METHOD INTERNAL CreateCommandPayloadLog
VAR_IN_OUT
  /// Robot assignment of function
  AxesGroup : AxesGroup; 
END_VAR
VAR 
  /// internal index for loops
 _idx : DINT;
END_VAR
// Create log entry for Parameter start
CreateLogMessage      ( Timestamp   := AxesGroup.InternalData.SystemTime,
                        MessageType := MessageType.CMD,
                        Severity    := Severity.DEBUG,
                        MessageCode := 0,
                        MessageText := 'Create command payload with the following parameter(s) :');

// Create log entry for Mode
CreateLogMessagePara1 ( Timestamp   := AxesGroup.InternalData.SystemTime,
                        MessageType := MessageType.CMD,
                        Severity    := Severity.DEBUG,
                        MessageCode := 0,
                        MessageText := 'Command.Mode = {1}',
                        Para1       :=  SPLINE_MODE_TO_STRING(_command.Mode));

// Create log entry for SplineID
CreateLogMessagePara1 ( Timestamp   := AxesGroup.InternalData.SystemTime,
                        MessageType := MessageType.CMD,
                        Severity    := Severity.DEBUG,
                        MessageCode := 0,
                        MessageText := 'Command.SplineID = {1}',
                        Para1       :=  SINT_TO_STRING(_command.SplineID));

// Create log entry for SplineData[x]
FOR _idx := 1 TO RobotLibraryParameter.SPLINE_DATA_MAX
DO
  // Create log entry for VelocityRate
  CreateLogMessagePara2 ( Timestamp   := AxesGroup.InternalData.SystemTime,
                          MessageType := MessageType.CMD,
                          Severity    := Severity.DEBUG,
                          MessageCode := 0,
                          MessageText := 'Command.SplineData[{2}].VelocityRate = {1}',
                          Para1       :=  UINT_TO_STRING(_command.SplineData[_idx].VelocityRate),
                          Para2       :=  DINT_TO_STRING(_idx));

  // Create log entry for AccelerationRate
  CreateLogMessagePara2 ( Timestamp   := AxesGroup.InternalData.SystemTime,
                          MessageType := MessageType.CMD,
                          Severity    := Severity.DEBUG,
                          MessageCode := 0,
                          MessageText := 'Command.SplineData[{2}].AccelerationRate = {1}',
                          Para1       :=  UINT_TO_STRING(_command.SplineData[_idx].AccelerationRate),
                          Para2       :=  DINT_TO_STRING(_idx));

  // Create log entry for DecelerationRate
  CreateLogMessagePara2 ( Timestamp   := AxesGroup.InternalData.SystemTime,
                          MessageType := MessageType.CMD,
                          Severity    := Severity.DEBUG,
                          MessageCode := 0,
                          MessageText := 'Command.SplineData[{2}].DecelerationRate = {1}',
                          Para1       :=  UINT_TO_STRING(_command.SplineData[_idx].DecelerationRate),
                          Para2       :=  DINT_TO_STRING(_idx));
                          
  // Create log entry for JerkRate
  CreateLogMessagePara2 ( Timestamp   := AxesGroup.InternalData.SystemTime,
                          MessageType := MessageType.CMD,
                          Severity    := Severity.DEBUG,
                          MessageCode := 0,
                          MessageText := 'Command.SplineData[{2}].JerkRate = {1}',
                          Para1       :=  UINT_TO_STRING(_command.SplineData[_idx].JerkRate),
                          Para2       :=  DINT_TO_STRING(_idx));

                          
  // Create log entry for ToolNo
  CreateLogMessagePara2 ( Timestamp   := AxesGroup.InternalData.SystemTime,
                          MessageType := MessageType.CMD,
                          Severity    := Severity.DEBUG,
                          MessageCode := 0,
                          MessageText := 'Command.SplineData[{2}].ToolNo = {1}',
                          Para1       :=  USINT_TO_STRING(_command.SplineData[_idx].ToolNo),
                          Para2       :=  DINT_TO_STRING(_idx));
  
  // Create log entry for FrameNo
  CreateLogMessagePara2 ( Timestamp   := AxesGroup.InternalData.SystemTime,
                          MessageType := MessageType.CMD,
                          Severity    := Severity.DEBUG,
                          MessageCode := 0,
                          MessageText := 'Command.SplineData[{2}].FrameNo = {1}',
                          Para1       :=  USINT_TO_STRING(_command.SplineData[_idx].FrameNo),
                          Para2       :=  DINT_TO_STRING(_idx));
                          
  // Create log entry for Position.X
  CreateLogMessagePara2 ( Timestamp   := AxesGroup.InternalData.SystemTime,
                          MessageType := MessageType.CMD,
                          Severity    := Severity.DEBUG,
                          MessageCode := 0,
                          MessageText := 'Command.SplineData[{2}].Position.X = {1}',
                          Para1       :=  REAL_TO_STRING(_command.SplineData[_idx].Position.X),
                          Para2       :=  DINT_TO_STRING(_idx));

  // Create log entry for Position.Y
  CreateLogMessagePara2 ( Timestamp   := AxesGroup.InternalData.SystemTime,
                          MessageType := MessageType.CMD,
                          Severity    := Severity.DEBUG,
                          MessageCode := 0,
                          MessageText := 'Command.SplineData[{2}].Position.Y = {1}',
                          Para1       :=  REAL_TO_STRING(_command.SplineData[_idx].Position.Y),
                          Para2       :=  DINT_TO_STRING(_idx));
                          
  // Create log entry for Position.Z
  CreateLogMessagePara2 ( Timestamp   := AxesGroup.InternalData.SystemTime,
                          MessageType := MessageType.CMD,
                          Severity    := Severity.DEBUG,
                          MessageCode := 0,
                          MessageText := 'Command.SplineData[{2}].Position.Z = {1}',
                          Para1       :=  REAL_TO_STRING(_command.SplineData[_idx].Position.Z),
                          Para2       :=  DINT_TO_STRING(_idx));

  // Create log entry for Position.Rx
  CreateLogMessagePara2 ( Timestamp   := AxesGroup.InternalData.SystemTime,
                          MessageType := MessageType.CMD,
                          Severity    := Severity.DEBUG,
                          MessageCode := 0,
                          MessageText := 'Command.SplineData[{2}].Position.Rx = {1}',
                          Para1       :=  REAL_TO_STRING(_command.SplineData[_idx].Position.Rx),
                          Para2       :=  DINT_TO_STRING(_idx));
                          
  // Create log entry for Position.Ry
  CreateLogMessagePara2 ( Timestamp   := AxesGroup.InternalData.SystemTime,
                          MessageType := MessageType.CMD,
                          Severity    := Severity.DEBUG,
                          MessageCode := 0,
                          MessageText := 'Command.SplineData[{2}].Position.Ry = {1}',
                          Para1       :=  REAL_TO_STRING(_command.SplineData[_idx].Position.Ry),
                          Para2       :=  DINT_TO_STRING(_idx));
                          
  // Create log entry for Position.Rz
  CreateLogMessagePara2 ( Timestamp   := AxesGroup.InternalData.SystemTime,
                          MessageType := MessageType.CMD,
                          Severity    := Severity.DEBUG,
                          MessageCode := 0,
                          MessageText := 'Command.SplineData[{2}].Position.Rz = {1}',
                          Para1       :=  REAL_TO_STRING(_command.SplineData[_idx].Position.Rz),
                          Para2       :=  DINT_TO_STRING(_idx));

  // Create log entry for Position.Config
  CreateLogMessagePara2 ( Timestamp   := AxesGroup.InternalData.SystemTime,
                          MessageType := MessageType.CMD,
                          Severity    := Severity.DEBUG,
                          MessageCode := 0,
                          MessageText := 'Command.SplineData[{2}].Position.Config = {1}',
                          Para1       :=  ARM_CONFIG_TO_STRING(_command.SplineData[_idx].Position.Config),
                          Para2       :=  DINT_TO_STRING(_idx));

  // Create log entry for Position.TurnNumber[0]
  CreateLogMessagePara2 ( Timestamp   := AxesGroup.InternalData.SystemTime,
                          MessageType := MessageType.CMD,
                          Severity    := Severity.DEBUG,
                          MessageCode := 0,
                          MessageText := 'Command.SplineData[{2}].Position.TurnNumber[0] = {1}',
                          Para1       :=  BYTE_TO_STRING(CombineHalfSints(HalfSintHi := _command.SplineData[_idx].Position.TurnNumber.J2Turns,
                                                                          HalfSintLo := _command.SplineData[_idx].Position.TurnNumber.J1Turns)),                          
                          Para2       :=  DINT_TO_STRING(_idx));

  // Create log entry for Position.TurnNumber[1]
  CreateLogMessagePara2 ( Timestamp   := AxesGroup.InternalData.SystemTime,
                          MessageType := MessageType.CMD,
                          Severity    := Severity.DEBUG,
                          MessageCode := 0,
                          MessageText := 'Command.SplineData[{2}].Position.TurnNumber[1] = {1}',
                          Para1       :=  BYTE_TO_STRING(CombineHalfSints(HalfSintHi := _command.SplineData[_idx].Position.TurnNumber.J4Turns,
                                                                          HalfSintLo := _command.SplineData[_idx].Position.TurnNumber.J3Turns)),                          
                          Para2       :=  DINT_TO_STRING(_idx));
                          
  // Create log entry for Position.TurnNumber[2]
  CreateLogMessagePara2 ( Timestamp   := AxesGroup.InternalData.SystemTime,
                          MessageType := MessageType.CMD,
                          Severity    := Severity.DEBUG,
                          MessageCode := 0,
                          MessageText := 'Command.SplineData[{2}].Position.TurnNumber[2] = {1}',
                          Para1       :=  BYTE_TO_STRING(CombineHalfSints(HalfSintHi := _command.SplineData[_idx].Position.TurnNumber.J6Turns,
                                                                          HalfSintLo := _command.SplineData[_idx].Position.TurnNumber.J5Turns)),                          
                          Para2       :=  DINT_TO_STRING(_idx));

  // Create log entry for Position.TurnNumber[3]
  CreateLogMessagePara2 ( Timestamp   := AxesGroup.InternalData.SystemTime,
                          MessageType := MessageType.CMD,
                          Severity    := Severity.DEBUG,
                          MessageCode := 0,
                          MessageText := 'Command.SplineData[{2}].Position.TurnNumber[3] = {1}',
                          Para1       :=  SINT_TO_STRING(_command.SplineData[_idx].Position.TurnNumber.E1Turns),                          
                          Para2       :=  DINT_TO_STRING(_idx));
                          
  // Create log entry for Position.E1
  CreateLogMessagePara2 ( Timestamp   := AxesGroup.InternalData.SystemTime,
                          MessageType := MessageType.CMD,
                          Severity    := Severity.DEBUG,
                          MessageCode := 0,
                          MessageText := 'Command.SplineData[{2}].Position.E1 = {1}',
                          Para1       :=  REAL_TO_STRING(_command.SplineData[_idx].Position.E1),
                          Para2       :=  DINT_TO_STRING(_idx));

  // Create log entry for MoveTime
  CreateLogMessagePara2 ( Timestamp   := AxesGroup.InternalData.SystemTime,
                          MessageType := MessageType.CMD,
                          Severity    := Severity.DEBUG,
                          MessageCode := 0,
                          MessageText := 'Command.SplineData[{2}].MoveTime = {1}',
                          Para1       :=  UINT_TO_STRING(_command.SplineData[_idx].MoveTime),
                          Para2       :=  DINT_TO_STRING(_idx));

  // Create log entry for Position.E2
  CreateLogMessagePara2 ( Timestamp   := AxesGroup.InternalData.SystemTime,
                          MessageType := MessageType.CMD,
                          Severity    := Severity.DEBUG,
                          MessageCode := 0,
                          MessageText := 'Command.SplineData[{2}].Position.E2 = {1}',
                          Para1       :=  REAL_TO_STRING(_command.SplineData[_idx].Position.E2),
                          Para2       :=  DINT_TO_STRING(_idx));

  // Create log entry for Position.E3
  CreateLogMessagePara2 ( Timestamp   := AxesGroup.InternalData.SystemTime,
                          MessageType := MessageType.CMD,
                          Severity    := Severity.DEBUG,
                          MessageCode := 0,
                          MessageText := 'Command.SplineData[{2}].Position.E3 = {1}',
                          Para1       :=  REAL_TO_STRING(_command.SplineData[_idx].Position.E3),
                          Para2       :=  DINT_TO_STRING(_idx));

  // Create log entry for Position.E4
  CreateLogMessagePara2 ( Timestamp   := AxesGroup.InternalData.SystemTime,
                          MessageType := MessageType.CMD,
                          Severity    := Severity.DEBUG,
                          MessageCode := 0,
                          MessageText := 'Command.SplineData[{2}].Position.E4 = {1}',
                          Para1       :=  REAL_TO_STRING(_command.SplineData[_idx].Position.E4),
                          Para2       :=  DINT_TO_STRING(_idx));
                          
  // Create log entry for Position.E5
  CreateLogMessagePara2 ( Timestamp   := AxesGroup.InternalData.SystemTime,
                          MessageType := MessageType.CMD,
                          Severity    := Severity.DEBUG,
                          MessageCode := 0,
                          MessageText := 'Command.SplineData[{2}].Position.E5 = {1}',
                          Para1       :=  REAL_TO_STRING(_command.SplineData[_idx].Position.E5),
                          Para2       :=  DINT_TO_STRING(_idx));
                          
  // Create log entry for Position.E6
  CreateLogMessagePara2 ( Timestamp   := AxesGroup.InternalData.SystemTime,
                          MessageType := MessageType.CMD,
                          Severity    := Severity.DEBUG,
                          MessageCode := 0,
                          MessageText := 'Command.SplineData[{2}].Position.E6 = {1}',
                          Para1       :=  REAL_TO_STRING(_command.SplineData[_idx].Position.E6),
                          Para2       :=  DINT_TO_STRING(_idx));
                          
END_FOR
END_METHOD

METHOD FB_init : BOOL
VAR_INPUT
  /// if TRUE, the retain variables are initialized (warm start / cold start)
  bInitRetains : BOOL; 
  /// if TRUE, the instance afterwards gets moved into the copy code (online change)
  bInCopyCode  : BOOL;  
END_VAR
MyType := 'MC_CreateSplineFB';

ExecMode := ExecutionMode.PARALLEL;
END_METHOD

METHOD PROTECTED OnCall
VAR_IN_OUT
  /// Robot assignment of function
  AxesGroup : AxesGroup; 
END_VAR
// call base implementation
SUPER^.OnCall(AxesGroup := AxesGroup);

CASE _stepCmd OF
  
  00:  IF ( _execute_R.Q )  
       THEN
         // Check function is supported and parameter are valid ?
         IF (( CheckFunctionSupported( AxesGroup := AxesGroup )) AND
             ( CheckParameterValid   ( AxesGroup := AxesGroup )))
         THEN      
           // set busy flag
           Busy := TRUE;
           // Reset command outputs
           SysDepMemSet(pDest := ADR(OutCmd), Value := 0, DataLen := SIZEOF(OutCmd));         
           // apply command parameter
          _parCmd := ParCmd;
           // init parameter sequence
          _command.ParSeq := 1;
           // create command data
           CommandData := CreateCommandPayload(AxesGroup := AxesGroup);
           // Add command to active command register
          _uniqueID := AxesGroup.Acyclic.ActiveCommandRegister.AddCmd( pCommandFB := ADR(THIS^ ));     
           // set timeout
           SetTimeout(PT := _timeoutCmd, rTimer := _timerCmd);
           // inc step counter
          _stepCmd := _stepCmd + 1;
         END_IF 
       END_IF
     

  01:  // Wait for responce received
       IF ( _responseReceived )
       THEN
         // reset response received flag
        _responseReceived := FALSE;

         CASE  _response.State 
         OF
           CmdMessageState.BUFFERED : CommandBuffered := TRUE;
           CmdMessageState.DONE     : Done            := TRUE;
           CmdMessageState.ERROR    : Error           := TRUE;
         END_CASE
                
         // Done, Aborted or Error ?
         IF (_response.State >= CmdMessageState.DONE )
         THEN
           // Reset Busy flag
           Busy := FALSE;
           // set timeout
           SetTimeout(PT := _timeoutCmd, rTimer := _timerCmd);
           // inc step counter
          _stepCmd := _stepCmd + 1; 
         END_IF
       END_IF


  02: IF ( NOT Execute)
      THEN
        Reset(); 
      END_IF     

ELSE
  // invalid step
  ErrorID := RobotLibraryEvents.ERR_INVALID_STEP;
END_CASE


// Reset FB
IF ( NOT Execute )
THEN
  Reset();
END_IF
END_METHOD

METHOD INTERNAL ParseResponsePayload : DINT
VAR_INPUT
  /// Response data
  ResponseData : RobotLibraryRecvDataFB;
  /// Timestamp
  Timestamp    : SystemTime;  
END_VAR
// Table 6-755: Received CMD payload (RC to PLC) of "CreateSpline"
// --------------------------
// Header
// --------------------------
// Byte 00 : USINT   - ParSeq | State     
// Byte 01 : SINT    - AlarmMessageSeverity    
// Byte 02 : UINT    - AlarmMessageCode HB
// Byte 03 :         - AlarmMessageCode LB
// call base implementation to parse the header from payload buffer
ResponseData.PayloadPtr := SUPER^.ParseResponsePayload(ResponseData := ResponseData, Timestamp := Timestamp);

// copy parsed header to response
_response.ParSeq               := _rspHeader.ParSeq;
_response.State                := _rspHeader.State;
_response.AlarmMessageSeverity := _rspHeader.AlarmMessageSeverity;
_response.AlarmMessageCode     := _rspHeader.AlarmMessageCode;

// Create logging
ParseResponsePayloadLog(ResponseData := ResponseData, Timestamp := Timestamp);
END_METHOD

METHOD INTERNAL ParseResponsePayloadLog
VAR_INPUT
  /// Response data
  ResponseData : RobotLibraryRecvDataFB;
  /// Timestamp
  Timestamp    : SystemTime;  
END_VAR
// Create log entry for Parameter start
CreateLogMessage      ( Timestamp   := Timestamp,
                        MessageType := MessageType.CMD,
                        Severity    := Severity.DEBUG,
                        MessageCode := 0,
                        MessageText := 'Parsed the following parameter(s) from response data:');
                        
// Create log entry for no parameter 
CreateLogMessage      ( Timestamp   := Timestamp,
                        MessageType := MessageType.CMD,
                        Severity    := Severity.DEBUG,
                        MessageCode := 0,
                        MessageText := 'This command has no parameter to parse...');
END_METHOD

METHOD PROTECTED Reset : DINT
VAR_INPUT
END_VAR
Reset := SUPER^.Reset();

Done               := FALSE;
Busy               := FALSE;
CommandBuffered    := FALSE;
END_METHOD

END_FUNCTION_BLOCK

// Library/POUs/Spline/MC_DeleteSpline/MC_DeleteSplineFB
/// Delete spline previously created on RC
FUNCTION_BLOCK MC_DeleteSplineFB EXTENDS RobotLibraryBaseExecuteFB
// ------------------------------------------------------------------------- 
//  SRCI Robot Library                                                
// ------------------------------------------------------------------------- 
//                                                                           
//  Object:      DeleteSplineFB                                       
//  Author:      Thorsten Brach                                                
//  Date:        2024-06-01
//
//  Description:                                              
//   
//                                                                           
//  Copyright: 
//    (C) 2024 Thorsten Brach. All rights reserved                                                                                                                                            
//             Licensed under the LGPL-3.0 license.
//                                                                           
//  Disclaimer:                                                                           
//    This project is provided without any guarantee and can be used for   
//    private and commercial purposes. Any use is at the user’s 
//    own risk and responsibility.
//
// -------------------------------------------------------------------------
VAR_INPUT
  /// command parameter 
  ParCmd          : DeleteSplineParCmd;
END_VAR
VAR_OUTPUT
  /// Command is transferred and confirmed by the RC
  CommandBuffered : BOOL;
  /// command results
  OutCmd          : DeleteSplineOutCmd;     
END_VAR

VAR
  /// internal copy of command parameter 
 _parCmd          : DeleteSplineParCmd;
  /// command data to send
 _command         : DeleteSplineSendData;
  /// response data received
 _response        : DeleteSplineRecvData;      
END_VAR

SUPER^(AxesGroup := AxesGroup);

METHOD PROTECTED CheckFunctionSupported : BOOL
VAR_IN_OUT
  /// Robot assignment of function
  AxesGroup : AxesGroup; 
END_VAR
CheckFunctionSupported := AxesGroup.InternalData.RCSupportedFunctions.DeleteSpline;

IF ( NOT CheckFunctionSupported )
THEN
  // call base implementation for set error and create log entry
  SUPER^.CheckFunctionSupported(AxesGroup := AxesGroup);
END_IF
END_METHOD

METHOD PROTECTED CheckParameterChanged : BOOL
VAR_IN_OUT
  /// Robot assignment of function
  AxesGroup    : AxesGroup; 
END_VAR
// Check ParCmd Size is > 0, because MemCmp does not work correctly with size = 0
IF (SIZEOF(ParCmd) = 0) 
THEN 
  RETURN;
END_IF

// compare memory 
_parameterChanged := ( SysDepMemCmp(pData1 := ADR(ParCmd), pData2 := ADR(_parCmd), DataLen := SIZEOF(ParCmd)) <> RobotLibraryConstants.OK );

// check parameter valid ?
_parameterValid   := CheckParameterValid( AxesGroup := AxesGroup );

IF ((  _parameterChanged        )  AND 
    (  _parameterValid          )) OR
    (  _parameterUpdateInternal )  
THEN  
  // reset internal flag for send parameter update
 _parameterUpdateInternal := FALSE;
  // update internal copy of parameters 
 _parCmd := ParCmd;
  // inc parameter sequence
 _command.ParSeq := _command.ParSeq + 1;
  // update command data  
  CommandData := CreateCommandPayload(AxesGroup := AxesGroup); // ( Access via reference to rCommandFB in ACR )
  // notify active command register 
  AxesGroup.Acyclic.ActiveCommandRegister.NotifyParameterChanged := _uniqueID;
END_IF
END_METHOD

METHOD INTERNAL CreateCommandPayload : RobotLibrarySendDataFB
VAR_IN_OUT
  /// Robot assignment of function
  AxesGroup : AxesGroup; 
END_VAR
// Table 6-760: Sent CMD payload (PLC to RC) of "DeleteSpline"
// --------------------------
// Header
// --------------------------
// Byte 00 : UINT  - Type HB     
// Byte 01 :       - Type LB    
// Byte 02 : USINT - Reserve | ExecutionMode
// Byte 03 : USINT - ParSeq  | Priority
// --------------------------
// Datablock
// --------------------------
 // Byte 04 : SINT  SplineID;
// set command parameter 
_command.CmdTyp   :=  CmdType.DeleteSpline;
_command.ExecMode :=  ExecMode;
_command.ParSeq   := _command.ParSeq;
_command.Priority :=  Priority;
_command.SplineID := _parCmd.SplineID;

// copy command data to header
_cmdHeader := _command;
// call base implementation to copy header to payload buffer
CreateCommandPayload := SUPER^.CreateCommandPayload(AxesGroup := AxesGroup);

// add command.SplineID
CreateCommandPayload.AddSint(_command.SplineID);

// Create logging
CreateCommandPayloadLog(AxesGroup := AxesGroup);
END_METHOD

METHOD INTERNAL CreateCommandPayloadLog
VAR_IN_OUT
  /// Robot assignment of function
  AxesGroup : AxesGroup; 
END_VAR
// Create log entry for Parameter start
CreateLogMessage      ( Timestamp   := AxesGroup.InternalData.SystemTime,
                        MessageType := MessageType.CMD,
                        Severity    := Severity.DEBUG,
                        MessageCode := 0,
                        MessageText := 'Create command payload with the following parameter(s) :');
  
// Create log entry for SplineID
CreateLogMessagePara1 ( Timestamp   := AxesGroup.InternalData.SystemTime,
                        MessageType := MessageType.CMD,
                        Severity    := Severity.DEBUG,
                        MessageCode := 0,
                        MessageText := 'Command.SplineID = {1}',
                        Para1       :=  SINT_TO_STRING(_command.SplineID));
END_METHOD

METHOD FB_init : BOOL
VAR_INPUT
  /// if TRUE, the retain variables are initialized (warm start / cold start)
  bInitRetains : BOOL; 
  /// if TRUE, the instance afterwards gets moved into the copy code (online change)
  bInCopyCode  : BOOL;  
END_VAR
MyType := 'MC_DeleteSplineFB';

ExecMode := ExecutionMode.PARALLEL;
END_METHOD

METHOD PROTECTED OnCall
VAR_IN_OUT
  /// Robot assignment of function
  AxesGroup : AxesGroup; 
END_VAR
// call base implementation
SUPER^.OnCall(AxesGroup := AxesGroup);

CASE _stepCmd OF
  
  00:  IF ( _execute_R.Q )  
       THEN
         // Check function is supported and parameter are valid ?
         IF (( CheckFunctionSupported( AxesGroup := AxesGroup )) AND
             ( CheckParameterValid   ( AxesGroup := AxesGroup )))
         THEN      
           // set busy flag
           Busy := TRUE;
           // Reset command outputs
           SysDepMemSet(pDest := ADR(OutCmd), Value := 0, DataLen := SIZEOF(OutCmd));         
           // apply command parameter
          _parCmd := ParCmd;
           // init parameter sequence
          _command.ParSeq := 1;
           // create command data
           CommandData := CreateCommandPayload(AxesGroup := AxesGroup);
           // Add command to active command register
          _uniqueID := AxesGroup.Acyclic.ActiveCommandRegister.AddCmd( pCommandFB := ADR(THIS^ ));     
           // set timeout
           SetTimeout(PT := _timeoutCmd, rTimer := _timerCmd);
           // inc step counter
          _stepCmd := _stepCmd + 1;
         END_IF 
       END_IF
     

  01:  // Wait for responce received
       IF ( _responseReceived )
       THEN
         // reset response received flag
        _responseReceived := FALSE;

         CASE  _response.State 
         OF
           CmdMessageState.BUFFERED : CommandBuffered := TRUE;
           CmdMessageState.DONE     : Done            := TRUE;
           CmdMessageState.ERROR    : Error           := TRUE;
         END_CASE
                
         // Done, Aborted or Error ?
         IF (_response.State >= CmdMessageState.DONE )
         THEN
           // Reset Busy flag
           Busy := FALSE;
           // set timeout
           SetTimeout(PT := _timeoutCmd, rTimer := _timerCmd);
           // inc step counter
          _stepCmd := _stepCmd + 1; 
         END_IF
       END_IF


  02: IF ( NOT Execute)
      THEN
        Reset(); 
      END_IF     

ELSE
  // invalid step
  ErrorID := RobotLibraryEvents.ERR_INVALID_STEP;
END_CASE


// Reset FB
IF ( NOT Execute )
THEN
  Reset(); 
END_IF
END_METHOD

METHOD INTERNAL ParseResponsePayload : DINT
VAR_INPUT
  /// Response data
  ResponseData : RobotLibraryRecvDataFB;
  /// Timestamp
  Timestamp    : SystemTime;  
END_VAR
// Table 6-761: Received CMD payload (RC to PLC) of "DeleteSpline"
// --------------------------
// Header
// --------------------------
// Byte 00 : USINT   - ParSeq | State     
// Byte 01 : SINT    - AlarmMessageSeverity    
// Byte 02 : UINT    - AlarmMessageCode HB
// Byte 03 :         - AlarmMessageCode LB
// call base implementation to parse the header from payload buffer
ResponseData.PayloadPtr := SUPER^.ParseResponsePayload(ResponseData := ResponseData, Timestamp := Timestamp);

// copy parsed header to response
_response.ParSeq               := _rspHeader.ParSeq;
_response.State                := _rspHeader.State;
_response.AlarmMessageSeverity := _rspHeader.AlarmMessageSeverity;
_response.AlarmMessageCode     := _rspHeader.AlarmMessageCode;

// Create logging
ParseResponsePayloadLog(ResponseData := ResponseData, Timestamp := Timestamp);
END_METHOD

METHOD INTERNAL ParseResponsePayloadLog
VAR_INPUT
  /// Response data
  ResponseData : RobotLibraryRecvDataFB;
  /// Timestamp
  Timestamp    : SystemTime;  
END_VAR
// Create log entry for Parameter start
CreateLogMessage      ( Timestamp   := Timestamp,
                        MessageType := MessageType.CMD,
                        Severity    := Severity.DEBUG,
                        MessageCode := 0,
                        MessageText := 'Parsed the following parameter(s) from response data:');
                        
// Create log entry for no parameter 
CreateLogMessage      ( Timestamp   := Timestamp,
                        MessageType := MessageType.CMD,
                        Severity    := Severity.DEBUG,
                        MessageCode := 0,
                        MessageText := 'This command has no parameter to parse...');
END_METHOD

METHOD PROTECTED Reset : DINT
VAR_INPUT
END_VAR
Reset := SUPER^.Reset();

Done               := FALSE;
Busy               := FALSE;
CommandBuffered    := FALSE;
END_METHOD

END_FUNCTION_BLOCK

// Library/POUs/Spline/MC_DynamicSpline/MC_DynamicSplineFB
/// Create and move spline on RC simultaneously
FUNCTION_BLOCK MC_DynamicSplineFB EXTENDS RobotLibraryBaseFB
// ------------------------------------------------------------------------- 
//  SRCI Robot Library                                                
// ------------------------------------------------------------------------- 
//                                                                           
//  Object:      DynamicSplineFB                                       
//  Author:      Thorsten Brach                                                
//  Date:        2024-06-01
//
//  Description:                                              
//   
//                                                                           
//  Copyright: 
//    (C) 2024 Thorsten Brach. All rights reserved                                                                                                                                            
//             Licensed under the LGPL-3.0 license.
//                                                                           
//  Disclaimer:                                                                           
//    This project is provided without any guarantee and can be used for   
//    private and commercial purposes. Any use is at the user’s 
//    own risk and responsibility.
//
// -------------------------------------------------------------------------
VAR_INPUT
  /// Start of the command at the rising edge
  Execute            : BOOL;
  /// Parameter which determines the behavior towards the previously sent and still active or buffered commands
  AbortingMode       : AbortingMode;
  /// Defines the target sequence in which the command will be executed
  SequenceFlag       : SequenceFlag;
  /// command parameter 
  ParCmd             : DynamicSplineParCmd;
END_VAR
VAR_OUTPUT
  /// FB is being processed
  Busy               : BOOL;
  /// Command is transferred and confirmed by the RC
  CommandBuffered    : BOOL;
  /// Function is enabled and new input values will be transmitted.
  Enabled            : BOOL;
  /// The command takes control of the motion of the according axis group
  Active             : BOOL;
  /// The command was aborted by another command.
  CommandAborted     : BOOL;
  /// TRUE, while command is interrupted during execution and can be continued.
  CommandInterrupted : BOOL;
  /// Receiving of input parameter values has been acknowledged by RC
  ParameterAccepted  : BOOL;
  /// command results
  OutCmd             : DynamicSplineOutCmd;     
END_VAR

VAR
  /// internal copy of command parameter 
 _parCmd             : DynamicSplineParCmd;
  /// command data to send
 _command            : DynamicSplineSendData;
  /// response data received
 _response           : DynamicSplineRecvData;      
END_VAR

SUPER^(AxesGroup := AxesGroup);

METHOD PROTECTED CheckFunctionSupported : BOOL
VAR_IN_OUT
  /// Robot assignment of function
  AxesGroup : AxesGroup; 
END_VAR
CheckFunctionSupported := AxesGroup.InternalData.RCSupportedFunctions.DynamicSpline;

IF ( NOT CheckFunctionSupported )
THEN
  // call base implementation for set error and create log entry
  SUPER^.CheckFunctionSupported(AxesGroup := AxesGroup);
END_IF
END_METHOD

METHOD PROTECTED CheckParameterChanged : BOOL
VAR_IN_OUT
  /// Robot assignment of function
  AxesGroup    : AxesGroup; 
END_VAR
// Check ParCmd Size is > 0, because MemCmp does not work correctly with size = 0
IF (SIZEOF(ParCmd) = 0) 
THEN 
  RETURN;
END_IF

// compare memory 
_parameterChanged := ( SysDepMemCmp(pData1 := ADR(ParCmd), pData2 := ADR(_parCmd), DataLen := SIZEOF(ParCmd)) <> RobotLibraryConstants.OK );

// check parameter valid ?
_parameterValid   := CheckParameterValid( AxesGroup := AxesGroup );

IF ((  _parameterChanged        )  AND 
    (  _parameterValid          )) OR
    (  _parameterUpdateInternal )  
THEN  
  // reset internal flag for send parameter update
 _parameterUpdateInternal := FALSE;
  // update internal copy of parameters 
 _parCmd := ParCmd;
  // inc parameter sequence
 _command.ParSeq := _command.ParSeq + 1;
  // update command data  
  CommandData := CreateCommandPayload(AxesGroup := AxesGroup); // ( Access via reference to rCommandFB in ACR )
  // notify active command register 
  AxesGroup.Acyclic.ActiveCommandRegister.NotifyParameterChanged := _uniqueID;
  // Reset parameter accepted flag
  ParameterAccepted := FALSE;  
END_IF
END_METHOD

METHOD INTERNAL CreateCommandPayload : RobotLibrarySendDataFB
VAR_IN_OUT
  /// Robot assignment of function
  AxesGroup : AxesGroup; 
END_VAR
// Table 6-772: Sent CMD payload (PLC to RC) of "DynamicSpline"
// --------------------------
// Header
// --------------------------
// Byte 00 : UINT  - Type HB     
// Byte 01 :       - Type LB    
// Byte 02 : USINT - Reserve | ExecutionMode
// Byte 03 : USINT - ParSeq  | Priority
// --------------------------
// Datablock
// --------------------------
// Byte 00 : UINT  Type;
// Byte 01 :       Type;
// Byte 02 : USINT Reserved ExecutionMode;
// Byte 03 : USINT ParSeq Priority;
// Byte 04 : UINT  Mode;
// Byte 05 : USINT BlendingMode;
// Byte 06 : REAL  BlendingParameter[0];
// Byte 07 :       BlendingParameter[0];
// Byte 08 :       BlendingParameter[0];
// Byte 09 :       BlendingParameter[0];
// Byte 10 : REAL  BlendingParameter[1];
// Byte 11 :       BlendingParameter[1];
// Byte 12 :       BlendingParameter[1];
// Byte 13 :       BlendingParameter[1];
// Byte 14 : UINT  Time;
// Byte 15 :       Time;
// Byte 16 : INT   StartPosition;
// Byte 17 :       StartPosition;
// Byte 18 : UINT  SplineData.VelocityRate;
// Byte 19 :       SplineData.VelocityRate;
// Byte 20 : UINT  SplineData.AccelerationRate;
// Byte 21 :       SplineData.AccelerationRate;
// Byte 22 : UINT  SplineData.DecelerationRate;
// Byte 23 :       SplineData.DecelerationRate;
// Byte 24 : UINT  SplineData.JerkRate;
// Byte 25 :       SplineData.JerkRate;
// Byte 26 : USINT SplineData.ToolNo;
// Byte 27 : USINT SplineData.FrameNo;
// Byte 28 : REAL  SplineData.X;
// Byte 29 :       SplineData.X;
// Byte 30 :       SplineData.X;
// Byte 31 :       SplineData.X;
// Byte 32 : REAL  SplineData.Y;
// Byte 33 :       SplineData.Y;
// Byte 34 :       SplineData.Y;
// Byte 35 :       SplineData.Y;
// Byte 36 : REAL  SplineData.Z;
// Byte 37 :       SplineData.Z;
// Byte 38 :       SplineData.Z;
// Byte 39 :       SplineData.Z;
// Byte 40 : REAL  SplineData.RX;
// Byte 41 :       SplineData.RX;
// Byte 42 :       SplineData.RX;
// Byte 43 :       SplineData.RX;
// Byte 44 : REAL  SplineData.RY;
// Byte 45 :       SplineData.RY;
// Byte 46 :       SplineData.RY;
// Byte 47 :       SplineData.RY;
// Byte 48 : REAL  SplineData.RZ;
// Byte 49 :       SplineData.RZ;
// Byte 50 :       SplineData.RZ;
// Byte 51 :       SplineData.RZ;
// Byte 52 : BYTE  - - - - - W E S;
// Byte 53 : BYTE  Reserved;
// Byte 54 : BYTE  SplineData.TurnNumber[0];
// Byte 55 : BYTE  SplineData.TurnNumber[1];
// Byte 56 : BYTE  SplineData.TurnNumber[2];
// Byte 57 : BYTE  SplineData.TurnNumber[3];
// Byte 58 : REAL  SplineData.E1;
// Byte 59 :       SplineData.E1;
// Byte 60 :       SplineData.E1;
// Byte 61 :       SplineData.E1;
// Byte 62 : UINT  SplineData.Time;
// Byte 63 :       SplineData.Time;
// Byte 64 : REAL  SplineData.E2;
// Byte 65 :       SplineData.E2;
// Byte 66 :       SplineData.E2;
// Byte 67 :       SplineData.E2;
// Byte 68 : REAL  SplineData.E3;
// Byte 69 :       SplineData.E3;
// Byte 70 :       SplineData.E3;
// Byte 71 :       SplineData.E3;
// Byte 72 : REAL  SplineData.E4;
// Byte 73 :       SplineData.E4;
// Byte 74 :       SplineData.E4;
// Byte 75 :       SplineData.E4;
// Byte 76 : REAL  SplineData.E5;
// Byte 77 :       SplineData.E5;
// Byte 78 :       SplineData.E5;
// Byte 79 :       SplineData.E5;
// Byte 80 : REAL  SplineData.E6;
// Byte 81 :       SplineData.E6;
// Byte 82 :       SplineData.E6;
// Byte 83 :       SplineData.E6;
VAR
  /// internal index for loops
  _idx : DINT;
END_VAR
// set command parameter 
_command.CmdTyp            :=  CmdType.DynamicSpline;
_command.ExecMode          :=  ExecMode;
_command.ParSeq            := _command.ParSeq;
_command.Priority          :=  Priority;
_command.Mode              := _parCmd.Mode;
_command.BlendingMode      := _parCmd.BlendingMode;
_command.BlendingParameter := _parCmd.BlendingParameter;
_command.MoveTime          := TIME_TO_UINT(_parCmd.MoveTime);
_command.StartPosition     := _parCmd.StartPosition;

FOR _idx := 1 TO RobotLibraryParameter.SPLINE_DATA_MAX
DO
  _command.SplineData[_idx].VelocityRate     := REAL_TO_PERCENT_UINT(_parCmd.SplineData[_idx].VelocityRate     , IsOptional := FALSE);
  _command.SplineData[_idx].AccelerationRate := REAL_TO_PERCENT_UINT(_parCmd.SplineData[_idx].AccelerationRate , IsOptional := FALSE);
  _command.SplineData[_idx].DecelerationRate := REAL_TO_PERCENT_UINT(_parCmd.SplineData[_idx].DecelerationRate , IsOptional := TRUE );
  _command.SplineData[_idx].JerkRate         := REAL_TO_PERCENT_UINT(_parCmd.SplineData[_idx].JerkRate         , IsOptional := TRUE );
  _command.SplineData[_idx].ToolNo           :=              _parCmd.SplineData[_idx].ToolNo;
  _command.SplineData[_idx].FrameNo          :=              _parCmd.SplineData[_idx].FrameNo;
  _command.SplineData[_idx].MoveTime         := TIME_TO_UINT(_parCmd.SplineData[_idx].MoveTime);
END_FOR

// copy command data to header
_cmdHeader := _command;
// call base implementation to copy header to payload buffer
CreateCommandPayload := SUPER^.CreateCommandPayload(AxesGroup := AxesGroup);


// add command.Mode
CreateCommandPayload.AddUint(_command.Mode);
// add command.BlendingMode
CreateCommandPayload.AddUsint(_command.BlendingMode);
// add command.BlendingParameter[0]
CreateCommandPayload.AddReal(_command.BlendingParameter[0]);
// add command.BlendingParameter[1]
CreateCommandPayload.AddReal(_command.BlendingParameter[1]);
// add command.MoveTime
CreateCommandPayload.AddUint(_command.MoveTime);
// add command.StartPosition
CreateCommandPayload.AddInt(_command.StartPosition);


FOR _idx := 1 TO RobotLibraryParameter.SPLINE_DATA_MAX
DO
  // add command.VelocityRate
  CreateCommandPayload.AddUint(_command.SplineData[_idx].VelocityRate);
  // add command.AccelerationRate
  CreateCommandPayload.AddUint(_command.SplineData[_idx].AccelerationRate);
  // add command.DecelerationRate
  CreateCommandPayload.AddUint(_command.SplineData[_idx].DecelerationRate);
  // add command.JerkRate
  CreateCommandPayload.AddUint(_command.SplineData[_idx].JerkRate);
  // add command.ToolNo
  CreateCommandPayload.AddUsint(_command.SplineData[_idx].ToolNo);
  // add command.FrameNo
  CreateCommandPayload.AddUsint(_command.SplineData[_idx].FrameNo);
  // add command.SplineData[_idx].Position.X
  CreateCommandPayload.AddReal(_command.SplineData[_idx].Position.X);
  // add command.SplineData[_idx].Position.Y
  CreateCommandPayload.AddReal(_command.SplineData[_idx].Position.Y);
  // add command.SplineData[_idx].Position.Z
  CreateCommandPayload.AddReal(_command.SplineData[_idx].Position.Z);
  // add command.SplineData[_idx].Position.Rx
  CreateCommandPayload.AddReal(_command.SplineData[_idx].Position.Rx);
  // add command.SplineData[_idx].Position.Ry
  CreateCommandPayload.AddReal(_command.SplineData[_idx].Position.Ry);
  // add command.SplineData[_idx].Position.Rz
  CreateCommandPayload.AddReal(_command.SplineData[_idx].Position.Rz);
  // add command.SplineData[_idx].Position.Config
  CreateCommandPayload.AddArmConfig(_command.SplineData[_idx].Position.Config);
  // add command.SplineData[_idx].Position.TurnNumber
  CreateCommandPayload.AddTurnNumber(_command.SplineData[_idx].Position.TurnNumber);
  // add command.SplineData[_idx].Position.E1
  CreateCommandPayload.AddReal(_command.SplineData[_idx].Position.E1);
  // add command.SplineData[_idx].MoveTime
  CreateCommandPayload.AddUint(_command.SplineData[_idx].MoveTime);  
  // add command.SplineData[_idx].Position.E2
  CreateCommandPayload.AddReal(_command.SplineData[_idx].Position.E2);
  // add command.SplineData[_idx].Position.E3
  CreateCommandPayload.AddReal(_command.SplineData[_idx].Position.E3);
  // add command.SplineData[_idx].Position.E4
  CreateCommandPayload.AddReal(_command.SplineData[_idx].Position.E4);
  // add command.SplineData[_idx].Position.E5
  CreateCommandPayload.AddReal(_command.SplineData[_idx].Position.E5);
  // add command.SplineData[_idx].Position.E6
  CreateCommandPayload.AddReal(_command.SplineData[_idx].Position.E6);
END_FOR

// Create logging
CreateCommandPayloadLog(AxesGroup := AxesGroup);
END_METHOD

METHOD INTERNAL CreateCommandPayloadLog
VAR_IN_OUT
  /// Robot assignment of function
  AxesGroup : AxesGroup; 
END_VAR
VAR 
  /// internal index for loops
 _idx : DINT;
END_VAR
// Create log entry for Parameter start
CreateLogMessage      ( Timestamp   := AxesGroup.InternalData.SystemTime,
                        MessageType := MessageType.CMD,
                        Severity    := Severity.DEBUG,
                        MessageCode := 0,
                        MessageText := 'Create command payload with the following parameter(s) :');

// Create log entry for Mode
CreateLogMessagePara1 ( Timestamp   := AxesGroup.InternalData.SystemTime,
                        MessageType := MessageType.CMD,
                        Severity    := Severity.DEBUG,
                        MessageCode := 0,
                        MessageText := 'Command.Mode = {1}',
                        Para1       :=  SPLINE_MODE_TO_STRING(_command.Mode));

// Create log entry for BlendingMode
CreateLogMessagePara1 ( Timestamp   := AxesGroup.InternalData.SystemTime,
                        MessageType := MessageType.CMD,
                        Severity    := Severity.DEBUG,
                        MessageCode := 0,
                        MessageText := 'Command.BlendingMode = {1}',
                        Para1       :=  BLENDING_MODE_TO_STRING(_command.BlendingMode));

// Create log entry for BlendingParameter[0]
CreateLogMessagePara1 ( Timestamp   := AxesGroup.InternalData.SystemTime,
                        MessageType := MessageType.CMD,
                        Severity    := Severity.DEBUG,
                        MessageCode := 0,
                        MessageText := 'Command.BlendingParameter[0] = {1}',
                        Para1       :=  REAL_TO_STRING(_command.BlendingParameter[0]));

// Create log entry for BlendingParameter[1]
CreateLogMessagePara1 ( Timestamp   := AxesGroup.InternalData.SystemTime,
                        MessageType := MessageType.CMD,
                        Severity    := Severity.DEBUG,
                        MessageCode := 0,
                        MessageText := 'Command.BlendingParameter[1] = {1}',
                        Para1       :=  REAL_TO_STRING(_command.BlendingParameter[1]));

// Create log entry for MoveTime
CreateLogMessagePara1 ( Timestamp   := AxesGroup.InternalData.SystemTime,
                        MessageType := MessageType.CMD,
                        Severity    := Severity.DEBUG,
                        MessageCode := 0,
                        MessageText := 'Command.MoveTime = {1}',
                        Para1       :=  REAL_TO_STRING(_command.MoveTime));

// Create log entry for StartPosition
CreateLogMessagePara1 ( Timestamp   := AxesGroup.InternalData.SystemTime,
                        MessageType := MessageType.CMD,
                        Severity    := Severity.DEBUG,
                        MessageCode := 0,
                        MessageText := 'Command.StartPosition = {1}',
                        Para1       :=  INT_TO_STRING(_command.StartPosition));

// Create log entry for SplineData[x]
FOR _idx := 1 TO RobotLibraryParameter.SPLINE_DATA_MAX
DO
  // Create log entry for VelocityRate
  CreateLogMessagePara2 ( Timestamp   := AxesGroup.InternalData.SystemTime,
                          MessageType := MessageType.CMD,
                          Severity    := Severity.DEBUG,
                          MessageCode := 0,
                          MessageText := 'Command.SplineData[{2}].VelocityRate = {1}',
                          Para1       :=  UINT_TO_STRING(_command.SplineData[_idx].VelocityRate),
                          Para2       :=  DINT_TO_STRING(_idx));

  // Create log entry for AccelerationRate
  CreateLogMessagePara2 ( Timestamp   := AxesGroup.InternalData.SystemTime,
                          MessageType := MessageType.CMD,
                          Severity    := Severity.DEBUG,
                          MessageCode := 0,
                          MessageText := 'Command.SplineData[{2}].AccelerationRate = {1}',
                          Para1       :=  UINT_TO_STRING(_command.SplineData[_idx].AccelerationRate),
                          Para2       :=  DINT_TO_STRING(_idx));

  // Create log entry for DecelerationRate
  CreateLogMessagePara2 ( Timestamp   := AxesGroup.InternalData.SystemTime,
                          MessageType := MessageType.CMD,
                          Severity    := Severity.DEBUG,
                          MessageCode := 0,
                          MessageText := 'Command.SplineData[{2}].DecelerationRate = {1}',
                          Para1       :=  UINT_TO_STRING(_command.SplineData[_idx].DecelerationRate),
                          Para2       :=  DINT_TO_STRING(_idx));
                          
  // Create log entry for JerkRate
  CreateLogMessagePara2 ( Timestamp   := AxesGroup.InternalData.SystemTime,
                          MessageType := MessageType.CMD,
                          Severity    := Severity.DEBUG,
                          MessageCode := 0,
                          MessageText := 'Command.SplineData[{2}].JerkRate = {1}',
                          Para1       :=  UINT_TO_STRING(_command.SplineData[_idx].JerkRate),
                          Para2       :=  DINT_TO_STRING(_idx));

                          
  // Create log entry for ToolNo
  CreateLogMessagePara2 ( Timestamp   := AxesGroup.InternalData.SystemTime,
                          MessageType := MessageType.CMD,
                          Severity    := Severity.DEBUG,
                          MessageCode := 0,
                          MessageText := 'Command.SplineData[{2}].ToolNo = {1}',
                          Para1       :=  USINT_TO_STRING(_command.SplineData[_idx].ToolNo),
                          Para2       :=  DINT_TO_STRING(_idx));
  
  // Create log entry for FrameNo
  CreateLogMessagePara2 ( Timestamp   := AxesGroup.InternalData.SystemTime,
                          MessageType := MessageType.CMD,
                          Severity    := Severity.DEBUG,
                          MessageCode := 0,
                          MessageText := 'Command.SplineData[{2}].FrameNo = {1}',
                          Para1       :=  USINT_TO_STRING(_command.SplineData[_idx].FrameNo),
                          Para2       :=  DINT_TO_STRING(_idx));
                          
  // Create log entry for Position.X
  CreateLogMessagePara2 ( Timestamp   := AxesGroup.InternalData.SystemTime,
                          MessageType := MessageType.CMD,
                          Severity    := Severity.DEBUG,
                          MessageCode := 0,
                          MessageText := 'Command.SplineData[{2}].Position.X = {1}',
                          Para1       :=  REAL_TO_STRING(_command.SplineData[_idx].Position.X),
                          Para2       :=  DINT_TO_STRING(_idx));

  // Create log entry for Position.Y
  CreateLogMessagePara2 ( Timestamp   := AxesGroup.InternalData.SystemTime,
                          MessageType := MessageType.CMD,
                          Severity    := Severity.DEBUG,
                          MessageCode := 0,
                          MessageText := 'Command.SplineData[{2}].Position.Y = {1}',
                          Para1       :=  REAL_TO_STRING(_command.SplineData[_idx].Position.Y),
                          Para2       :=  DINT_TO_STRING(_idx));
                          
  // Create log entry for Position.Z
  CreateLogMessagePara2 ( Timestamp   := AxesGroup.InternalData.SystemTime,
                          MessageType := MessageType.CMD,
                          Severity    := Severity.DEBUG,
                          MessageCode := 0,
                          MessageText := 'Command.SplineData[{2}].Position.Z = {1}',
                          Para1       :=  REAL_TO_STRING(_command.SplineData[_idx].Position.Z),
                          Para2       :=  DINT_TO_STRING(_idx));

  // Create log entry for Position.Rx
  CreateLogMessagePara2 ( Timestamp   := AxesGroup.InternalData.SystemTime,
                          MessageType := MessageType.CMD,
                          Severity    := Severity.DEBUG,
                          MessageCode := 0,
                          MessageText := 'Command.SplineData[{2}].Position.Rx = {1}',
                          Para1       :=  REAL_TO_STRING(_command.SplineData[_idx].Position.Rx),
                          Para2       :=  DINT_TO_STRING(_idx));
                          
  // Create log entry for Position.Ry
  CreateLogMessagePara2 ( Timestamp   := AxesGroup.InternalData.SystemTime,
                          MessageType := MessageType.CMD,
                          Severity    := Severity.DEBUG,
                          MessageCode := 0,
                          MessageText := 'Command.SplineData[{2}].Position.Ry = {1}',
                          Para1       :=  REAL_TO_STRING(_command.SplineData[_idx].Position.Ry),
                          Para2       :=  DINT_TO_STRING(_idx));
                          
  // Create log entry for Position.Rz
  CreateLogMessagePara2 ( Timestamp   := AxesGroup.InternalData.SystemTime,
                          MessageType := MessageType.CMD,
                          Severity    := Severity.DEBUG,
                          MessageCode := 0,
                          MessageText := 'Command.SplineData[{2}].Position.Rz = {1}',
                          Para1       :=  REAL_TO_STRING(_command.SplineData[_idx].Position.Rz),
                          Para2       :=  DINT_TO_STRING(_idx));

  // Create log entry for Position.Config
  CreateLogMessagePara2 ( Timestamp   := AxesGroup.InternalData.SystemTime,
                          MessageType := MessageType.CMD,
                          Severity    := Severity.DEBUG,
                          MessageCode := 0,
                          MessageText := 'Command.SplineData[{2}].Position.Config = {1}',
                          Para1       :=  ARM_CONFIG_TO_STRING(_command.SplineData[_idx].Position.Config),
                          Para2       :=  DINT_TO_STRING(_idx));

  // Create log entry for Position.TurnNumber[0]
  CreateLogMessagePara2 ( Timestamp   := AxesGroup.InternalData.SystemTime,
                          MessageType := MessageType.CMD,
                          Severity    := Severity.DEBUG,
                          MessageCode := 0,
                          MessageText := 'Command.SplineData[{2}].Position.TurnNumber[0] = {1}',
                          Para1       :=  BYTE_TO_STRING(CombineHalfSints(HalfSintHi := _command.SplineData[_idx].Position.TurnNumber.J2Turns,
                                                                          HalfSintLo := _command.SplineData[_idx].Position.TurnNumber.J1Turns)),                          
                          Para2       :=  DINT_TO_STRING(_idx));

  // Create log entry for Position.TurnNumber[1]
  CreateLogMessagePara2 ( Timestamp   := AxesGroup.InternalData.SystemTime,
                          MessageType := MessageType.CMD,
                          Severity    := Severity.DEBUG,
                          MessageCode := 0,
                          MessageText := 'Command.SplineData[{2}].Position.TurnNumber[1] = {1}',
                          Para1       :=  BYTE_TO_STRING(CombineHalfSints(HalfSintHi := _command.SplineData[_idx].Position.TurnNumber.J4Turns,
                                                                          HalfSintLo := _command.SplineData[_idx].Position.TurnNumber.J3Turns)),                          
                          Para2       :=  DINT_TO_STRING(_idx));
                          
  // Create log entry for Position.TurnNumber[2]
  CreateLogMessagePara2 ( Timestamp   := AxesGroup.InternalData.SystemTime,
                          MessageType := MessageType.CMD,
                          Severity    := Severity.DEBUG,
                          MessageCode := 0,
                          MessageText := 'Command.SplineData[{2}].Position.TurnNumber[2] = {1}',
                          Para1       :=  BYTE_TO_STRING(CombineHalfSints(HalfSintHi := _command.SplineData[_idx].Position.TurnNumber.J6Turns,
                                                                          HalfSintLo := _command.SplineData[_idx].Position.TurnNumber.J5Turns)),                          
                          Para2       :=  DINT_TO_STRING(_idx));

  // Create log entry for Position.TurnNumber[3]
  CreateLogMessagePara2 ( Timestamp   := AxesGroup.InternalData.SystemTime,
                          MessageType := MessageType.CMD,
                          Severity    := Severity.DEBUG,
                          MessageCode := 0,
                          MessageText := 'Command.SplineData[{2}].Position.TurnNumber[3] = {1}',
                          Para1       :=  SINT_TO_STRING(_command.SplineData[_idx].Position.TurnNumber.E1Turns),                          
                          Para2       :=  DINT_TO_STRING(_idx));
                          
  // Create log entry for Position.E1
  CreateLogMessagePara2 ( Timestamp   := AxesGroup.InternalData.SystemTime,
                          MessageType := MessageType.CMD,
                          Severity    := Severity.DEBUG,
                          MessageCode := 0,
                          MessageText := 'Command.SplineData[{2}].Position.E1 = {1}',
                          Para1       :=  REAL_TO_STRING(_command.SplineData[_idx].Position.E1),
                          Para2       :=  DINT_TO_STRING(_idx));

  // Create log entry for MoveTime
  CreateLogMessagePara2 ( Timestamp   := AxesGroup.InternalData.SystemTime,
                          MessageType := MessageType.CMD,
                          Severity    := Severity.DEBUG,
                          MessageCode := 0,
                          MessageText := 'Command.SplineData[{2}].MoveTime = {1}',
                          Para1       :=  UINT_TO_STRING(_command.SplineData[_idx].MoveTime),
                          Para2       :=  DINT_TO_STRING(_idx));

  // Create log entry for Position.E2
  CreateLogMessagePara2 ( Timestamp   := AxesGroup.InternalData.SystemTime,
                          MessageType := MessageType.CMD,
                          Severity    := Severity.DEBUG,
                          MessageCode := 0,
                          MessageText := 'Command.SplineData[{2}].Position.E2 = {1}',
                          Para1       :=  REAL_TO_STRING(_command.SplineData[_idx].Position.E2),
                          Para2       :=  DINT_TO_STRING(_idx));

  // Create log entry for Position.E3
  CreateLogMessagePara2 ( Timestamp   := AxesGroup.InternalData.SystemTime,
                          MessageType := MessageType.CMD,
                          Severity    := Severity.DEBUG,
                          MessageCode := 0,
                          MessageText := 'Command.SplineData[{2}].Position.E3 = {1}',
                          Para1       :=  REAL_TO_STRING(_command.SplineData[_idx].Position.E3),
                          Para2       :=  DINT_TO_STRING(_idx));

  // Create log entry for Position.E4
  CreateLogMessagePara2 ( Timestamp   := AxesGroup.InternalData.SystemTime,
                          MessageType := MessageType.CMD,
                          Severity    := Severity.DEBUG,
                          MessageCode := 0,
                          MessageText := 'Command.SplineData[{2}].Position.E4 = {1}',
                          Para1       :=  REAL_TO_STRING(_command.SplineData[_idx].Position.E4),
                          Para2       :=  DINT_TO_STRING(_idx));
                          
  // Create log entry for Position.E5
  CreateLogMessagePara2 ( Timestamp   := AxesGroup.InternalData.SystemTime,
                          MessageType := MessageType.CMD,
                          Severity    := Severity.DEBUG,
                          MessageCode := 0,
                          MessageText := 'Command.SplineData[{2}].Position.E5 = {1}',
                          Para1       :=  REAL_TO_STRING(_command.SplineData[_idx].Position.E5),
                          Para2       :=  DINT_TO_STRING(_idx));
                          
  // Create log entry for Position.E6
  CreateLogMessagePara2 ( Timestamp   := AxesGroup.InternalData.SystemTime,
                          MessageType := MessageType.CMD,
                          Severity    := Severity.DEBUG,
                          MessageCode := 0,
                          MessageText := 'Command.SplineData[{2}].Position.E6 = {1}',
                          Para1       :=  REAL_TO_STRING(_command.SplineData[_idx].Position.E6),
                          Para2       :=  DINT_TO_STRING(_idx));
                          
END_FOR
END_METHOD

METHOD FB_init : BOOL
VAR_INPUT
  /// if TRUE, the retain variables are initialized (warm start / cold start)
  bInitRetains : BOOL; 
  /// if TRUE, the instance afterwards gets moved into the copy code (online change)
  bInCopyCode  : BOOL;  
END_VAR
MyType := 'MC_DynamicSplineFB';
END_METHOD

METHOD PROTECTED OnCall
VAR_IN_OUT
  /// Robot assignment of function
  AxesGroup : AxesGroup; 
END_VAR
// call base implementation
SUPER^.OnCall(AxesGroup := AxesGroup);

CASE _stepCmd OF
  
  00:  IF ( Execute )  
       THEN
         // Check function is supported and parameter are valid ?
         IF (( CheckFunctionSupported( AxesGroup := AxesGroup )) AND
             ( CheckParameterValid   ( AxesGroup := AxesGroup )))
         THEN      
           // set busy flag
           Busy := TRUE;
           // Reset command outputs
           SysDepMemSet(pDest := ADR(OutCmd), Value := 0, DataLen := SIZEOF(OutCmd));         
           // apply command parameter
          _parCmd := ParCmd;
           // init parameter sequence
          _command.ParSeq := 1;
           // create command data
           CommandData := CreateCommandPayload(AxesGroup := AxesGroup);
           // Add command to active command register
          _uniqueID := AxesGroup.Acyclic.ActiveCommandRegister.AddCmd( pCommandFB := ADR(THIS^ ));     
           // set timeout
           SetTimeout(PT := _timeoutCmd, rTimer := _timerCmd);
           // inc step counter
          _stepCmd := _stepCmd + 1; 
         END_IF
       END_IF
     

  01:  // Wait for responce received
       IF ( _responseReceived )
       THEN
         // reset response received flag
        _responseReceived := FALSE;

         CASE  _response.State 
         OF
           CmdMessageState.BUFFERED    : CommandBuffered    := TRUE;
           CmdMessageState.ABORTED     : CommandAborted     := TRUE;
           CmdMessageState.INTERRUPTED : CommandInterrupted := TRUE;           
           CmdMessageState.ERROR       : Error              := TRUE;
         END_CASE
                
         // Done, Aborted or Error ?
         IF (_response.State >= CmdMessageState.DONE )
         THEN
           // Update results
           OutCmd.SegmentProgress     := _response.SegmentProgress;
           OutCmd.RemainingDistance   := _response.RemainingDistance;
           OutCmd.Buffered            := _response.Buffered;
           OutCmd.Calculated          := _response.Calculated;
           OutCmd.ActiveIndex         := _response.ActiveIndex;
           OutCmd.TrajectoryCompleted := _response.TrajectoryCompleted;
           // set timeout
           SetTimeout(PT := _timeoutCmd, rTimer := _timerCmd);
           // inc step counter
          _stepCmd := _stepCmd + 1; 
         END_IF
       END_IF


  02: IF ( NOT Execute)
      THEN
        Reset();
      END_IF     

ELSE
  // invalid step
  ErrorID := RobotLibraryEvents.ERR_INVALID_STEP;
END_CASE


// Reset FB
IF ( NOT Execute )
THEN
 _uniqueId           := 0;
 _stepCmd            := 0;
  Busy               := FALSE;
  CommandBuffered    := FALSE;  
  CommandAborted     := FALSE;
  CommandInterrupted := FALSE;
  Error              := FALSE;
  ErrorID            := 0;
  WarningID          := 0;
  InfoID             := 0;  
END_IF
END_METHOD

METHOD INTERNAL ParseResponsePayload : DINT
VAR_INPUT
  /// Response data
  ResponseData : RobotLibraryRecvDataFB;
  /// Timestamp
  Timestamp    : SystemTime;  
END_VAR
// Table 6-773: Received CMD payload (RC to PLC) of "DynamicSpline"
// --------------------------
// Header
// --------------------------
// Byte 00 : USINT   - ParSeq | State     
// Byte 01 : SINT    - AlarmMessageSeverity    
// Byte 02 : UINT    - AlarmMessageCode HB
// Byte 03 :         - AlarmMessageCode LB
// --------------------------
// Datablock
// --------------------------
// Byte 04 : UINT    - Progress LW HB
// Byte 05 :         - Progress LW LB
// Byte 06 : REAL    - RemainingDistance HW HB
// Byte 07 :         - RemainingDistance HW LB
// Byte 08 :         - RemainingDistance LW HB
// Byte 09 :         - RemainingDistance LW LB
// Byte 10 : BOOL    - InClamping
// call base implementation to parse the header from payload buffer
ResponseData.PayloadPtr := SUPER^.ParseResponsePayload(ResponseData := ResponseData, Timestamp := Timestamp);

// copy parsed header to response
_response.ParSeq               := _rspHeader.ParSeq;
_response.State                := _rspHeader.State;
_response.AlarmMessageSeverity := _rspHeader.AlarmMessageSeverity;
_response.AlarmMessageCode     := _rspHeader.AlarmMessageCode;

// Get Response.Progress
_response.SegmentProgress := ResponseData.GetUint();
// Get Response.RemainingDistance
_response.RemainingDistance := ResponseData.GetReal();
// Get Response.Buffered
_response.Buffered := ResponseData.GetInt();
// Get Response.Calculated
_response.Calculated := ResponseData.GetInt();
// Get Response.ActiveIndex
_response.ActiveIndex := ResponseData.GetSint();
// Get Response.TrajectoryCompleted
_response.TrajectoryCompleted := ResponseData.GetBool();

// Create logging
ParseResponsePayloadLog(ResponseData := ResponseData, Timestamp := Timestamp);
END_METHOD

METHOD INTERNAL ParseResponsePayloadLog
VAR_INPUT
  /// Response data
  ResponseData : RobotLibraryRecvDataFB;
  /// Timestamp
  Timestamp    : SystemTime;  
END_VAR
// Create log entry for Parameter start
CreateLogMessage      ( Timestamp   := Timestamp,
                        MessageType := MessageType.CMD,
                        Severity    := Severity.DEBUG,
                        MessageCode := 0,
                        MessageText := 'Parsed the following parameter(s) from response data:');
                        
// Create log entry for SegmentProgress
CreateLogMessagePara1 ( Timestamp   := Timestamp,
                        MessageType := MessageType.CMD,
                        Severity    := Severity.DEBUG,
                        MessageCode := 0,
                        MessageText := 'Response.SegmentProgress = {1}',
                        Para1       :=  REAL_TO_STRING(_response.SegmentProgress));

// Create log entry for RemainingDistance
CreateLogMessagePara1 ( Timestamp   := Timestamp,
                        MessageType := MessageType.CMD,
                        Severity    := Severity.DEBUG,
                        MessageCode := 0,
                        MessageText := 'Response.RemainingDistance = {1}',
                        Para1       :=  REAL_TO_STRING(_response.RemainingDistance));

// Create log entry for Buffered
CreateLogMessagePara1 ( Timestamp   := Timestamp,
                        MessageType := MessageType.CMD,
                        Severity    := Severity.DEBUG,
                        MessageCode := 0,
                        MessageText := 'Response.Buffered = {1}',
                        Para1       :=  INT_TO_STRING(_response.Buffered));

// Create log entry for Calculated
CreateLogMessagePara1 ( Timestamp   := Timestamp,
                        MessageType := MessageType.CMD,
                        Severity    := Severity.DEBUG,
                        MessageCode := 0,
                        MessageText := 'Response.Calculated = {1}',
                        Para1       :=  INT_TO_STRING(_response.Calculated));

// Create log entry for ActiveIndex
CreateLogMessagePara1 ( Timestamp   := Timestamp,
                        MessageType := MessageType.CMD,
                        Severity    := Severity.DEBUG,
                        MessageCode := 0,
                        MessageText := 'Response.ActiveIndex = {1}',
                        Para1       :=  SINT_TO_STRING(_response.ActiveIndex));

// Create log entry for TrajectoryCompleted
CreateLogMessagePara1 ( Timestamp   := Timestamp,
                        MessageType := MessageType.CMD,
                        Severity    := Severity.DEBUG,
                        MessageCode := 0,
                        MessageText := 'Response.TrajectoryCompleted = {1}',
                        Para1       :=  BOOL_TO_STRING(_response.TrajectoryCompleted));
END_METHOD

METHOD PROTECTED Reset : DINT
VAR_INPUT
END_VAR
Reset := SUPER^.Reset();

Busy               := FALSE;
Active             := FALSE;
Enabled            := FALSE;
CommandBuffered    := FALSE;
CommandAborted     := FALSE;
CommandInterrupted := FALSE;
END_METHOD

END_FUNCTION_BLOCK

// Library/POUs/Spline/MC_MoveSpline/MC_MoveSplineFB
/// Move spline previously created on RC
FUNCTION_BLOCK MC_MoveSplineFB EXTENDS RobotLibraryBaseExecuteFB
// ------------------------------------------------------------------------- 
//  SRCI Robot Library                                                
// ------------------------------------------------------------------------- 
//                                                                           
//  Object:      MoveSplineFB                                       
//  Author:      Thorsten Brach                                                
//  Date:        2024-06-01
//
//  Description:                                              
//   
//                                                                           
//  Copyright: 
//    (C) 2024 Thorsten Brach. All rights reserved                                                                                                                                            
//             Licensed under the LGPL-3.0 license.
//                                                                           
//  Disclaimer:                                                                           
//    This project is provided without any guarantee and can be used for   
//    private and commercial purposes. Any use is at the user’s 
//    own risk and responsibility.
//
// -------------------------------------------------------------------------
VAR_INPUT
  ///Parameter which determines the behavior towards the previously sent and still active or buffered commands
  AbortingMode       : AbortingMode;
  /// Defines the target sequence in which the command will be executed
  SequenceFlag       : SequenceFlag;
  /// command parametre
  ParCmd             : MoveSplineParCmd;       
END_VAR
VAR_OUTPUT
  /// Command is transferred and confirmed by the RC
  CommandBuffered    : BOOL;
  /// The command takes control of the motion of the according axis group.
  Active             : BOOL;
  /// The command was aborted by another command
  CommandAborted     : BOOL;
  /// TRUE, while command is interrupted during execution and can be continued
  CommandInterrupted : BOOL;
  /// command outputs
  OutCmd             : MoveSplineOutCmd;       
END_VAR



VAR
  /// internal copy of command parameter 
 _parCmd             : MoveSplineParCmd;
  /// command data to send
 _command            : MoveSplineSendData;
  /// response data received
 _response           : MoveSplineRecvData;      
END_VAR

SUPER^(AxesGroup := AxesGroup);

METHOD PROTECTED CheckFunctionSupported : BOOL
VAR_IN_OUT
  /// Robot assignment of function
  AxesGroup : AxesGroup; 
END_VAR
CheckFunctionSupported := AxesGroup.InternalData.RCSupportedFunctions.MoveSpline;

IF ( NOT CheckFunctionSupported )
THEN
  // call base implementation for set error and create log entry
  SUPER^.CheckFunctionSupported(AxesGroup := AxesGroup);
END_IF
END_METHOD

METHOD PROTECTED CheckParameterChanged : BOOL
VAR_IN_OUT
  /// Robot assignment of function
  AxesGroup    : AxesGroup; 
END_VAR
// Check ParCmd Size is > 0, because MemCmp does not work correctly with size = 0
IF (SIZEOF(ParCmd) = 0) 
THEN 
  RETURN;
END_IF

// compare memory 
_parameterChanged := ( SysDepMemCmp(pData1 := ADR(ParCmd), pData2 := ADR(_parCmd), DataLen := SIZEOF(ParCmd)) <> RobotLibraryConstants.OK );

// check parameter valid ?
_parameterValid   := CheckParameterValid( AxesGroup := AxesGroup );

IF ((  _parameterChanged        )  AND 
    (  _parameterValid          )) OR
    (  _parameterUpdateInternal )  
THEN  
  // reset internal flag for send parameter update
 _parameterUpdateInternal := FALSE;
  // update internal copy of parameters 
 _parCmd := ParCmd;
  // inc parameter sequence
 _command.ParSeq := _command.ParSeq + 1;
  // update command data  
  CommandData := CreateCommandPayload(AxesGroup := AxesGroup); // ( Access via reference to rCommandFB in ACR )
  // notify active command register 
  AxesGroup.Acyclic.ActiveCommandRegister.NotifyParameterChanged := _uniqueID;
END_IF
END_METHOD

METHOD INTERNAL CreateCommandPayload : RobotLibrarySendDataFB
VAR_IN_OUT
  /// Robot assignment of function
  AxesGroup : AxesGroup; 
END_VAR
// Table 6-766: Sent CMD payload (PLC to RC) of "MoveSpline"
// --------------------------
// Header
// --------------------------
// Byte 00 : UINT  - Type HB     
// Byte 01 :       - Type LB    
// Byte 02 : USINT - Reserve | ExecutionMode
// Byte 03 : USINT - ParSeq  | Priority
// --------------------------
// Datablock
// --------------------------
// Byte 04 : SINT  SplineID;
// Byte 05 : USINT BlendingMode;
// Byte 06 : REAL  BlendingParameter[0];
// Byte 07 :       BlendingParameter[0];
// Byte 08 :       BlendingParameter[0];
// Byte 09 :       BlendingParameter[0];
// Byte 10 : REAL  BlendingParameter[1];
// Byte 11 :       BlendingParameter[1];
// Byte 12 :       BlendingParameter[1];
// Byte 13 :       BlendingParameter[1];
// Byte 14 : UINT  Time;
// Byte 15 :       Time;
// --------------------------
// set command parameter 
_command.CmdTyp            :=  CmdType.MoveSpline;
_command.ExecMode          :=  ExecMode;
_command.ParSeq            := _command.ParSeq;
_command.Priority          :=  Priority;
_command.SplineID          := _parCmd.SplineID;
_command.BlendingMode      := _parCmd.BlendingMode;
_command.BlendingParameter := _parCmd.BlendingParameter;
_command.MoveTime          := TIME_TO_UINT(_parCmd.MoveTime);


// copy command data to header
_cmdHeader := _command;
// call base implementation to copy header to payload buffer
CreateCommandPayload := SUPER^.CreateCommandPayload(AxesGroup := AxesGroup);

// add command.SplineID
CreateCommandPayload.AddSint(_command.SplineID);
// add command.BlendingMode
CreateCommandPayload.AddUsint(_command.BlendingMode);
// add command.BlendingParameter[0]
CreateCommandPayload.AddReal(_command.BlendingParameter[0]);
// add command.BlendingParameter[1]
CreateCommandPayload.AddReal(_command.BlendingParameter[1]);
// add command.MoveTime
CreateCommandPayload.AddUint(_command.MoveTime);

// Create logging
CreateCommandPayloadLog(AxesGroup := AxesGroup);
END_METHOD

METHOD INTERNAL CreateCommandPayloadLog
VAR_IN_OUT
  /// Robot assignment of function
  AxesGroup : AxesGroup; 
END_VAR
// Create log entry for Parameter start
CreateLogMessage      ( Timestamp   := AxesGroup.InternalData.SystemTime,
                        MessageType := MessageType.CMD,
                        Severity    := Severity.DEBUG,
                        MessageCode := 0,
                        MessageText := 'Create command payload with the following parameter(s) :');

// Create log entry for SplineID
CreateLogMessagePara1 ( Timestamp   := AxesGroup.InternalData.SystemTime,
                        MessageType := MessageType.CMD,
                        Severity    := Severity.DEBUG,
                        MessageCode := 0,
                        MessageText := 'Command.SplineID = {1}',
                        Para1       :=  SINT_TO_STRING(_command.SplineID));

// Create log entry for BlendingMode
CreateLogMessagePara1 ( Timestamp   := AxesGroup.InternalData.SystemTime,
                        MessageType := MessageType.CMD,
                        Severity    := Severity.DEBUG,
                        MessageCode := 0,
                        MessageText := 'Command.BlendingMode = {1}',
                        Para1       :=  BLENDING_MODE_TO_STRING(_command.BlendingMode));

// Create log entry for BlendingParameter[0]
CreateLogMessagePara1 ( Timestamp   := AxesGroup.InternalData.SystemTime,
                        MessageType := MessageType.CMD,
                        Severity    := Severity.DEBUG,
                        MessageCode := 0,
                        MessageText := 'Command.BlendingParameter[0] = {1}',
                        Para1       :=  REAL_TO_STRING(_command.BlendingParameter[0]));

// Create log entry for BlendingParameter[1]
CreateLogMessagePara1 ( Timestamp   := AxesGroup.InternalData.SystemTime,
                        MessageType := MessageType.CMD,
                        Severity    := Severity.DEBUG,
                        MessageCode := 0,
                        MessageText := 'Command.BlendingParameter[1] = {1}',
                        Para1       :=  REAL_TO_STRING(_command.BlendingParameter[1]));

// Create log entry for MoveTime
CreateLogMessagePara1 ( Timestamp   := AxesGroup.InternalData.SystemTime,
                        MessageType := MessageType.CMD,
                        Severity    := Severity.DEBUG,
                        MessageCode := 0,
                        MessageText := 'Command.MoveTime = {1}',
                        Para1       :=  REAL_TO_STRING(_command.MoveTime));
END_METHOD

METHOD FB_init : BOOL
VAR_INPUT
  /// if TRUE, the retain variables are initialized (warm start / cold start)
  bInitRetains : BOOL; 
  /// if TRUE, the instance afterwards gets moved into the copy code (online change)
  bInCopyCode  : BOOL;  
END_VAR
MyType := 'MC_MoveSplineFB';
END_METHOD

METHOD PROTECTED OnCall
VAR_IN_OUT
  /// Robot assignment of function
  AxesGroup : AxesGroup; 
END_VAR
// call base implementation
SUPER^.OnCall(AxesGroup := AxesGroup);

CASE _stepCmd OF
  
  00:  IF ( _execute_R.Q )  
       THEN
         // Check function is supported and parameter are valid ?
         IF (( CheckFunctionSupported( AxesGroup := AxesGroup )) AND
             ( CheckParameterValid   ( AxesGroup := AxesGroup )))
         THEN      
           // set busy flag
           Busy := TRUE;
           // Reset command outputs
           SysDepMemSet(pDest := ADR(OutCmd), Value := 0, DataLen := SIZEOF(OutCmd));         
           // apply command parameter
          _parCmd := ParCmd;
           // init parameter sequence
          _command.ParSeq := 1;
           // create command data
           CommandData := CreateCommandPayload(AxesGroup := AxesGroup);
           // Add command to active command register
          _uniqueID := AxesGroup.Acyclic.ActiveCommandRegister.AddCmd( pCommandFB := ADR(THIS^ ));     
           // set timeout
           SetTimeout(PT := _timeoutCmd, rTimer := _timerCmd);
           // inc step counter
          _stepCmd := _stepCmd + 1; 
         END_IF
       END_IF


  01:  // Wait for responce received
       IF ( _responseReceived )
       THEN
         // reset response received flag
        _responseReceived := FALSE;
         // reset Active flag
         Active := FALSE;
         
         CASE  _response.State 
         OF
           CmdMessageState.BUFFERED    : CommandBuffered    := TRUE;
           CmdMessageState.ACTIVE      : Active             := TRUE;
           CmdMessageState.INTERRUPTED : CommandInterrupted := TRUE;           
           CmdMessageState.DONE        : Done               := TRUE;           
           CmdMessageState.ABORTED     : CommandAborted     := TRUE;
           CmdMessageState.ERROR       : Error              := TRUE;
         END_CASE
                
         // Done, Aborted or Error ?
         IF (_response.State >= CmdMessageState.DONE )
         THEN
           // Reset Busy flag
           Busy := FALSE;
           // Update results
           OutCmd.ActualIndex       := 0; {warning 'ToDo'}
           OutCmd.Progress          := _response.Progress;
           OutCmd.RemainingDistance := _response.RemainingDistance;
           // set timeout
           SetTimeout(PT := _timeoutCmd, rTimer := _timerCmd);
           // inc step counter
          _stepCmd := _stepCmd + 1; 
         END_IF
       END_IF


  02: IF ( NOT Execute)
      THEN
        Reset(); 
      END_IF     

ELSE
  // invalid step
  ErrorID := RobotLibraryEvents.ERR_INVALID_STEP;
END_CASE


// Reset FB
IF ( NOT Execute )
THEN
  Reset();
END_IF
END_METHOD

METHOD INTERNAL ParseResponsePayload : DINT
VAR_INPUT
  /// Response data
  ResponseData : RobotLibraryRecvDataFB;
  /// Timestamp
  Timestamp    : SystemTime;  
END_VAR
// Table 6-767: Received CMD payload (RC to PLC) of "MoveSpline"
// --------------------------
// Header
// --------------------------
// Byte 00 : USINT   - ParSeq | State     
// Byte 01 : SINT    - AlarmMessageSeverity    
// Byte 02 : UINT    - AlarmMessageCode HB
// Byte 03 :         - AlarmMessageCode LB
// --------------------------
// Datablock
// --------------------------
// Byte 04 : UINT       - Progress HW HB
// Byte 05 :            - Progress HW LB
// Byte 06 : REAL       - RemainingDistance HW HB
// Byte 07 :            - RemainingDistance HW LB
// Byte 08 :            - RemainingDistance LW HB
// Byte 09 :            - RemainingDistance LW LB
// call base implementation to parse the header from payload buffer
ResponseData.PayloadPtr := SUPER^.ParseResponsePayload(ResponseData := ResponseData, Timestamp := Timestamp);

// copy parsed header to response
_response.ParSeq               := _rspHeader.ParSeq;
_response.State                := _rspHeader.State;
_response.AlarmMessageSeverity := _rspHeader.AlarmMessageSeverity;
_response.AlarmMessageCode     := _rspHeader.AlarmMessageCode;

// Get Response.Progress
_response.Progress := ResponseData.GetUint();
// Get Response.RemainingDistance
_response.RemainingDistance := ResponseData.GetReal();

// Create logging
ParseResponsePayloadLog(ResponseData := ResponseData, Timestamp := Timestamp);
END_METHOD

METHOD INTERNAL ParseResponsePayloadLog
VAR_INPUT
  /// Response data
  ResponseData : RobotLibraryRecvDataFB;
  /// Timestamp
  Timestamp    : SystemTime;  
END_VAR
// Create log entry for Parameter start
CreateLogMessage      ( Timestamp   := Timestamp,
                        MessageType := MessageType.CMD,
                        Severity    := Severity.DEBUG,
                        MessageCode := 0,
                        MessageText := 'Parsed the following parameter(s) from response data:');
                        
// Create log entry for Progress
CreateLogMessagePara1 ( Timestamp   := Timestamp,
                        MessageType := MessageType.CMD,
                        Severity    := Severity.DEBUG,
                        MessageCode := 0,
                        MessageText := 'Response.Progress = {1}',
                        Para1       :=  UINT_TO_STRING(_response.Progress));

// Create log entry for RemainingDistance
CreateLogMessagePara1 ( Timestamp   := Timestamp,
                        MessageType := MessageType.CMD,
                        Severity    := Severity.DEBUG,
                        MessageCode := 0,
                        MessageText := 'Response.RemainingDistance = {1}',
                        Para1       :=  REAL_TO_STRING(_response.RemainingDistance));
END_METHOD

METHOD PROTECTED Reset : DINT
VAR_INPUT
END_VAR
Reset := SUPER^.Reset();

Done               := FALSE;
Busy               := FALSE;
Active             := FALSE;
CommandBuffered    := FALSE;
CommandAborted     := FALSE;
CommandInterrupted := FALSE;
END_METHOD

END_FUNCTION_BLOCK

// Library/POUs/SuperImposing/MC_MoveSuperImposed/MC_MoveSuperImposedFB
/// Activate superimposed motion of TCP to defined motion
FUNCTION_BLOCK MC_MoveSuperImposedFB EXTENDS RobotLibraryBaseExecuteFB
// ------------------------------------------------------------------------- 
//  SRCI Robot Library                                                
// ------------------------------------------------------------------------- 
//                                                                           
//  Object:      MoveSuperImposedFB                                       
//  Author:      Thorsten Brach                                                
//  Date:        2024-06-01
//
//  Description:                                              
//   
//                                                                           
//  Copyright: 
//    (C) 2024 Thorsten Brach. All rights reserved                                                                                                                                            
//             Licensed under the LGPL-3.0 license.
//                                                                           
//  Disclaimer:                                                                           
//    This project is provided without any guarantee and can be used for   
//    private and commercial purposes. Any use is at the user’s 
//    own risk and responsibility.
//
// -------------------------------------------------------------------------
VAR_INPUT
  /// command parameter 
  ParCmd            : MoveSuperImposedParCmd;
END_VAR

VAR_OUTPUT
  /// Command is transferred and confirmed by the RC
  CommandBuffered   : BOOL;
  /// The command takes control of the motion of the according axis group
  Active            : BOOL;
  /// Receiving of input parameter values has been acknowledged by RC
  ParameterAccepted : BOOL;
  /// command outputs
  OutCmd            : MoveSuperImposedOutCmd;       
END_VAR



VAR
  /// internal copy of command parameter 
 _parCmd             : MoveSuperImposedParCmd;
  /// command data to send
 _command            : MoveSuperImposedSendData;
  /// response data received
 _response           : MoveSuperImposedRecvData;      
END_VAR

SUPER^(AxesGroup := AxesGroup);

METHOD PROTECTED CheckFunctionSupported : BOOL
VAR_IN_OUT
  /// Robot assignment of function
  AxesGroup : AxesGroup; 
END_VAR
CheckFunctionSupported := AxesGroup.InternalData.RCSupportedFunctions.MoveSuperImposed;

IF ( NOT CheckFunctionSupported )
THEN
  // call base implementation for set error and create log entry
  SUPER^.CheckFunctionSupported(AxesGroup := AxesGroup);
END_IF
END_METHOD

METHOD PROTECTED CheckParameterChanged : BOOL
VAR_IN_OUT
  /// Robot assignment of function
  AxesGroup    : AxesGroup; 
END_VAR
// Check ParCmd Size is > 0, because MemCmp does not work correctly with size = 0
IF (SIZEOF(ParCmd) = 0) 
THEN 
  RETURN;
END_IF

// compare memory 
_parameterChanged := ( SysDepMemCmp(pData1 := ADR(ParCmd), pData2 := ADR(_parCmd), DataLen := SIZEOF(ParCmd)) <> RobotLibraryConstants.OK );

// check parameter valid ?
_parameterValid   := CheckParameterValid( AxesGroup := AxesGroup );

IF ((  _parameterChanged        )  AND 
    (  _parameterValid          )) OR
    (  _parameterUpdateInternal )  
THEN  
  // reset internal flag for send parameter update
 _parameterUpdateInternal := FALSE;
  // update internal copy of parameters 
 _parCmd := ParCmd;
  // inc parameter sequence
 _command.ParSeq := _command.ParSeq + 1;
  // update command data  
  CommandData := CreateCommandPayload(AxesGroup := AxesGroup); // ( Access via reference to rCommandFB in ACR )
  // notify active command register 
  AxesGroup.Acyclic.ActiveCommandRegister.NotifyParameterChanged := _uniqueID;
  // Reset parameter accepted flag
  ParameterAccepted := FALSE;  
END_IF
END_METHOD

METHOD INTERNAL CreateCommandPayload : RobotLibrarySendDataFB
VAR_IN_OUT
  /// Robot assignment of function
  AxesGroup : AxesGroup; 
END_VAR
// Table 6-464: Sent CMD payload (PLC to RC) of "MoveSuperImposed"
// --------------------------
// Header
// --------------------------
// Byte 00 : UINT  - Type HB     
// Byte 01 :       - Type LB    
// Byte 02 : USINT - Reserve | ExecutionMode
// Byte 03 : USINT - ParSeq  | Priority
// --------------------------
// Datablock
// --------------------------
// Byte 00 : UINT  Type;
// Byte 01 :       Type;
// Byte 02 : USINT Reserved ExecutionMode;
// Byte 03 : USINT ParSeq Priority;
// Byte 04 : SINT  EmitterID[0];
// Byte 05 : SINT  EmitterID[1];
// Byte 06 : SINT  EmitterID[2];
// Byte 07 : SINT  EmitterID[3];
// Byte 08 : SINT  ListenerID;
// Byte 09 : BYTE  Reserved;
// Byte 10 : UINT  VelocityRate;
// Byte 11 :       VelocityRate;
// Byte 12 : UINT  AccelerationRate;
// Byte 13 :       AccelerationRate;
// Byte 14 : UINT  DecelerationRate;
// Byte 15 :       DecelerationRate;
// Byte 16 : UINT  JerkRate;
// Byte 17 :       JerkRate;
// Byte 18 : USINT ToolNo;
// Byte 19 : USINT FrameNo;
// Byte 20 : REAL  Offset.X;
// Byte 21 :       Offset.X;
// Byte 22 :       Offset.X;
// Byte 23 :       Offset.X;
// Byte 24 : REAL  Offset.Y;
// Byte 25 :       Offset.Y;
// Byte 26 :       Offset.Y;
// Byte 27 :       Offset.Y;
// Byte 28 : REAL  Offset.Z;
// Byte 29 :       Offset.Z;
// Byte 30 :       Offset.Z;
// Byte 31 :       Offset.Z;
// Byte 32 : REAL  Offset.RX;
// Byte 33 :       Offset.RX;
// Byte 34 :       Offset.RX;
// Byte 35 :       Offset.RX;
// Byte 36 : REAL  Offset.RY;
// Byte 37 :       Offset.RY;
// Byte 38 :       Offset.RY;
// Byte 39 :       Offset.RY;
// Byte 40 : REAL  Offset.RZ;
// Byte 41 :       Offset.RZ;
// Byte 42 :       Offset.RZ;
// Byte 43 :       Offset.RZ;
// Byte 44 : BYTE  - - - - - W E S;
// Byte 45 : BYTE  Reserved;
// Byte 46 : BYTE  Offset.TurnNumber[0];
// Byte 47 : BYTE  Offset.TurnNumber[1];
// Byte 48 : BYTE  Offset.TurnNumber[2];
// Byte 49 : BYTE  Offset.TurnNumber[3];
// Byte 50 : REAL  Offset.E1;
// Byte 51 :       Offset.E1;
// Byte 52 :       Offset.E1;
// Byte 53 :       Offset.E1;
// Byte 54 : USINT ReferenceType;
// Byte 55 : BYTE  Reserved;
// Byte 56 : REAL  Offset.E2;
// Byte 57 :       Offset.E2;
// Byte 58 :       Offset.E2;
// Byte 59 :       Offset.E2;
// Byte 60 : REAL  Offset.E3;
// Byte 61 :       Offset.E3;
// Byte 62 :       Offset.E3;
// Byte 63 :       Offset.E3;
// Byte 64 : REAL  Offset.E4;
// Byte 65 :       Offset.E4;
// Byte 66 :       Offset.E4;
// Byte 67 :       Offset.E4;
// Byte 68 : REAL  Offset.E5;
// Byte 69 :       Offset.E5;
// Byte 70 :       Offset.E5;
// Byte 71 :       Offset.E5;
// Byte 72 : REAL  Offset.E6;
// Byte 73 :       Offset.E6;
// Byte 74 :       Offset.E6;
// Byte 75 :       Offset.E6;
// --------------------------
// set command parameter 
_command.CmdTyp               :=  CmdType.MoveSuperImposed;
_command.ExecMode             :=  ExecMode;
_command.ParSeq               := _command.ParSeq;
_command.Priority             :=  Priority;
_command.EmitterID            := _parCmd.EmitterID;
_command.ListenerID           := _parCmd.ListenerID;
_command.Reserve              :=  0;
_command.VelocityDiffRate     :=  REAL_TO_PERCENT_UINT(_parCmd.VelocityDiffRate     , IsOptional := FALSE);
_command.AccelerationDiffRate :=  REAL_TO_PERCENT_UINT(_parCmd.AccelerationDiffRate , IsOptional := FALSE);
_command.DecelerationDiffRate :=  REAL_TO_PERCENT_UINT(_parCmd.DecelerationDiffRate , IsOptional := TRUE );
_command.JerkDiffRate         :=  REAL_TO_PERCENT_UINT(_parCmd.JerkDiffRate         , IsOptional := TRUE );
_command.ToolNo               := _parCmd.ToolNo;
_command.FrameNo              := _parCmd.FrameNo;
_command.Offset               := _parCmd.Offset;
_command.ReferenceType        := _parCmd.ReferenceType;
_command.Reserve2             := 0;


// copy command data to header
_cmdHeader := _command;
// call base implementation to copy header to payload buffer
CreateCommandPayload := SUPER^.CreateCommandPayload(AxesGroup := AxesGroup);

// add command.EmitterID[0]
CreateCommandPayload.AddSint(_command.EmitterID[0]);
// add command.EmitterID[1]
CreateCommandPayload.AddSint(_command.EmitterID[1]);
// add command.EmitterID[2]
CreateCommandPayload.AddSint(_command.EmitterID[2]);
// add command.EmitterID[3]
CreateCommandPayload.AddSint(_command.EmitterID[3]);
// add command.ListenerID
CreateCommandPayload.AddSint(_command.ListenerID);
// add command.Reserve
CreateCommandPayload.AddByte(_command.Reserve);
// add command.VelocityDiffRate
CreateCommandPayload.AddUint(_command.VelocityDiffRate);
// add command.AccelerationDiffRate
CreateCommandPayload.AddUint(_command.AccelerationDiffRate);
// add command.DecelerationDiffRate
CreateCommandPayload.AddUint(_command.DecelerationDiffRate);
// add command.JerkDiffRate
CreateCommandPayload.AddUint(_command.JerkDiffRate);
// add command.ToolNo
CreateCommandPayload.AddUsint(_command.ToolNo);
// add command.FrameNo
CreateCommandPayload.AddUsint(_command.FrameNo);
// add command.Offset.X
CreateCommandPayload.AddReal(_command.Offset.X);
// add command.Offset.Y
CreateCommandPayload.AddReal(_command.Offset.Y);
// add command.Offset.Z
CreateCommandPayload.AddReal(_command.Offset.Z);
// add command.Offset.Rx
CreateCommandPayload.AddReal(_command.Offset.Rx);
// add command.Offset.Ry
CreateCommandPayload.AddReal(_command.Offset.Ry);
// add command.Offset.Rz
CreateCommandPayload.AddReal(_command.Offset.Rz);
// add command.Offset.Config
CreateCommandPayload.AddArmConfig(_command.Offset.Config);
// add command.Offset.TurnNumber
CreateCommandPayload.AddTurnNumber(_command.Offset.TurnNumber);
// add command.Offset.E1
CreateCommandPayload.AddReal(_command.Offset.E1);
// add command.ReferenceType
CreateCommandPayload.AddUsint(_command.ReferenceType);
// add command.Reserve2
CreateCommandPayload.AddByte(_command.Reserve2);
// add command.Offset.E2
CreateCommandPayload.AddReal(_command.Offset.E2);
// add command.Offset.E3
CreateCommandPayload.AddReal(_command.Offset.E3);
// add command.Offset.E4
CreateCommandPayload.AddReal(_command.Offset.E4);
// add command.Offset.E5
CreateCommandPayload.AddReal(_command.Offset.E5);
// add command.Offset.E6
CreateCommandPayload.AddReal(_command.Offset.E6);

// Create logging
CreateCommandPayloadLog(AxesGroup := AxesGroup);
END_METHOD

METHOD INTERNAL CreateCommandPayloadLog
VAR_IN_OUT
  /// Robot assignment of function
  AxesGroup : AxesGroup; 
END_VAR
VAR 
  /// internal index for loops
 _idx : DINT;
END_VAR

// Byte 20 : REAL  Offset.X;
// Byte 21 :       Offset.X;
// Byte 22 :       Offset.X;
// Byte 23 :       Offset.X;
// Byte 24 : REAL  Offset.Y;
// Byte 25 :       Offset.Y;
// Byte 26 :       Offset.Y;
// Byte 27 :       Offset.Y;
// Byte 28 : REAL  Offset.Z;
// Byte 29 :       Offset.Z;
// Byte 30 :       Offset.Z;
// Byte 31 :       Offset.Z;
// Byte 32 : REAL  Offset.RX;
// Byte 33 :       Offset.RX;
// Byte 34 :       Offset.RX;
// Byte 35 :       Offset.RX;
// Byte 36 : REAL  Offset.RY;
// Byte 37 :       Offset.RY;
// Byte 38 :       Offset.RY;
// Byte 39 :       Offset.RY;
// Byte 40 : REAL  Offset.RZ;
// Byte 41 :       Offset.RZ;
// Byte 42 :       Offset.RZ;
// Byte 43 :       Offset.RZ;
// Byte 44 : BYTE  - - - - - W E S;
// Byte 45 : BYTE  Reserved;
// Byte 46 : BYTE  Offset.TurnNumber[0];
// Byte 47 : BYTE  Offset.TurnNumber[1];
// Byte 48 : BYTE  Offset.TurnNumber[2];
// Byte 49 : BYTE  Offset.TurnNumber[3];
// Byte 50 : REAL  Offset.E1;
// Byte 51 :       Offset.E1;
// Byte 52 :       Offset.E1;
// Byte 53 :       Offset.E1;
// Byte 54 : USINT ReferenceType;
// Byte 55 : BYTE  Reserved;
// Byte 56 : REAL  Offset.E2;
// Byte 57 :       Offset.E2;
// Byte 58 :       Offset.E2;
// Byte 59 :       Offset.E2;
// Byte 60 : REAL  Offset.E3;
// Byte 61 :       Offset.E3;
// Byte 62 :       Offset.E3;
// Byte 63 :       Offset.E3;
// Byte 64 : REAL  Offset.E4;
// Byte 65 :       Offset.E4;
// Byte 66 :       Offset.E4;
// Byte 67 :       Offset.E4;
// Byte 68 : REAL  Offset.E5;
// Byte 69 :       Offset.E5;
// Byte 70 :       Offset.E5;
// Byte 71 :       Offset.E5;
// Byte 72 : REAL  Offset.E6;
// Byte 73 :       Offset.E6;
// Byte 74 :       Offset.E6;
// Byte 75 :       Offset.E6;
// Create log entry for Parameter start
CreateLogMessage      ( Timestamp   := AxesGroup.InternalData.SystemTime,
                        MessageType := MessageType.CMD,
                        Severity    := Severity.DEBUG,
                        MessageCode := 0,
                        MessageText := 'Create command payload with the following parameter(s) :');
  
// Create log entry for EmitterID[x]
FOR _idx := 0 TO 3
DO
  CreateLogMessagePara2 ( Timestamp   := AxesGroup.InternalData.SystemTime,
                          MessageType := MessageType.CMD,
                          Severity    := Severity.DEBUG,
                          MessageCode := 0,
                          MessageText := 'Command.EmitterID[{2}] = {1}',
                          Para1       :=  SINT_TO_STRING(_command.EmitterID[_idx]),
                          Para2       :=  DINT_TO_STRING(_idx));
END_FOR

// Create log entry for ListenerID
CreateLogMessagePara1 ( Timestamp   := AxesGroup.InternalData.SystemTime,
                        MessageType := MessageType.CMD,
                        Severity    := Severity.DEBUG,
                        MessageCode := 0,
                        MessageText := 'Command.ListenerID = {1}',
                        Para1       :=  SINT_TO_STRING(_command.ListenerID));
                        
// Create log entry for Reserve
CreateLogMessagePara1 ( Timestamp   := AxesGroup.InternalData.SystemTime,
                        MessageType := MessageType.CMD,
                        Severity    := Severity.DEBUG,
                        MessageCode := 0,
                        MessageText := 'Command.Reserve = {1}',
                        Para1       :=  BYTE_TO_STRING(_command.Reserve));

// Create log entry for VelocityDiffRate
CreateLogMessagePara1 ( Timestamp   := AxesGroup.InternalData.SystemTime,
                        MessageType := MessageType.CMD,
                        Severity    := Severity.DEBUG,
                        MessageCode := 0,
                        MessageText := 'Command.VelocityDiffRate = {1}',
                        Para1       :=  UINT_TO_STRING(_command.VelocityDiffRate));

// Create log entry for AccelerationDiffRate
CreateLogMessagePara1 ( Timestamp   := AxesGroup.InternalData.SystemTime,
                        MessageType := MessageType.CMD,
                        Severity    := Severity.DEBUG,
                        MessageCode := 0,
                        MessageText := 'Command.AccelerationDiffRate = {1}',
                        Para1       :=  UINT_TO_STRING(_command.AccelerationDiffRate));
                        
// Create log entry for DecelerationDiffRate
CreateLogMessagePara1 ( Timestamp   := AxesGroup.InternalData.SystemTime,
                        MessageType := MessageType.CMD,
                        Severity    := Severity.DEBUG,
                        MessageCode := 0,
                        MessageText := 'Command.DecelerationDiffRate = {1}',
                        Para1       :=  UINT_TO_STRING(_command.DecelerationDiffRate));

// Create log entry for JerkDiffRate
CreateLogMessagePara1 ( Timestamp   := AxesGroup.InternalData.SystemTime,
                        MessageType := MessageType.CMD,
                        Severity    := Severity.DEBUG,
                        MessageCode := 0,
                        MessageText := 'Command.JerkDiffRate = {1}',
                        Para1       :=  UINT_TO_STRING(_command.JerkDiffRate));

// Create log entry for ToolNo
CreateLogMessagePara1 ( Timestamp   := AxesGroup.InternalData.SystemTime,
                        MessageType := MessageType.CMD,
                        Severity    := Severity.DEBUG,
                        MessageCode := 0,
                        MessageText := 'Command.ToolNo = {1}',
                        Para1       :=  USINT_TO_STRING(_command.ToolNo));

// Create log entry for FrameNo
CreateLogMessagePara1 ( Timestamp   := AxesGroup.InternalData.SystemTime,
                        MessageType := MessageType.CMD,
                        Severity    := Severity.DEBUG,
                        MessageCode := 0,
                        MessageText := 'Command.FrameNo = {1}',
                        Para1       :=  USINT_TO_STRING(_command.FrameNo));

// Create log entry for Offset.X
CreateLogMessagePara1 ( Timestamp   := AxesGroup.InternalData.SystemTime,
                        MessageType := MessageType.CMD,
                        Severity    := Severity.DEBUG,
                        MessageCode := 0,
                        MessageText := 'Command.Offset.X = {1}',
                        Para1       :=  REAL_TO_STRING(_command.Offset.X));

// Create log entry for Offset.Y
CreateLogMessagePara1 ( Timestamp   := AxesGroup.InternalData.SystemTime,
                        MessageType := MessageType.CMD,
                        Severity    := Severity.DEBUG,
                        MessageCode := 0,
                        MessageText := 'Command.Offset.Y = {1}',
                        Para1       :=  REAL_TO_STRING(_command.Offset.Y));

